// Mitsubishi GX Works2 project: 축   PLC: Q02/Q02H

PROGRAM MAIN
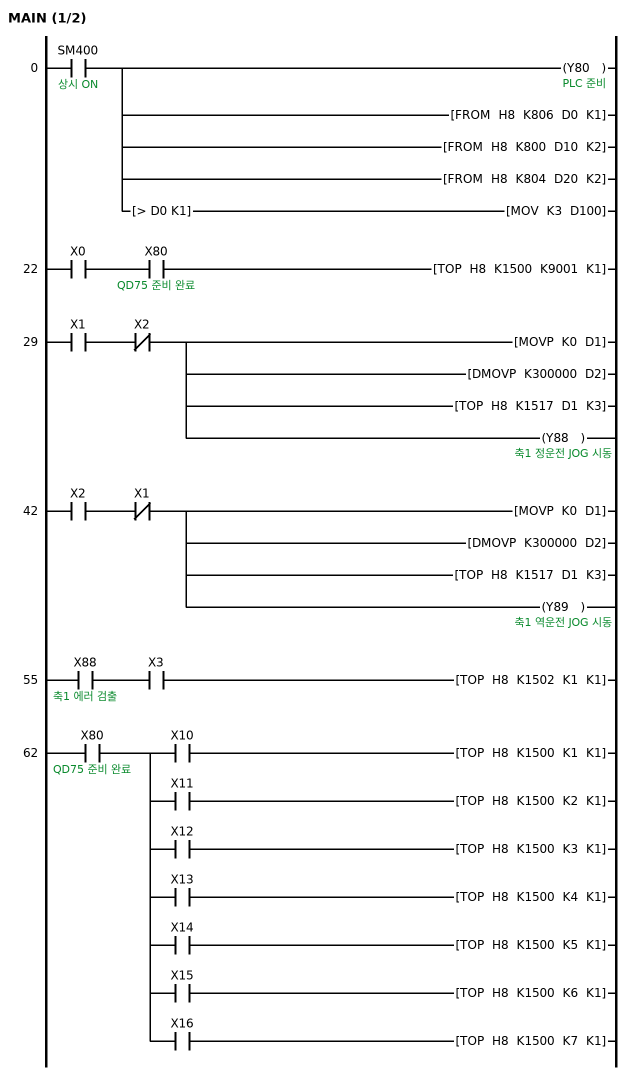
0     LD      SM400  ; 상시 ON
      OUT     Y80  ; PLC 준비
      FROM    H8 K806 D0 K1
      FROM    H8 K800 D10 K2
      FROM    H8 K804 D20 K2
      AND>    D0 K1
      MOV     K3 D100
22    LD      X0
      AND     X80  ; QD75 준비 완료
      TOP     H8 K1500 K9001 K1
29    LD      X1
      ANI     X2
      MOVP    K0 D1
      DMOVP   K300000 D2
      TOP     H8 K1517 D1 K3
      OUT     Y88  ; 축1 정운전 JOG 시동
42    LD      X2
      ANI     X1
      MOVP    K0 D1
      DMOVP   K300000 D2
      TOP     H8 K1517 D1 K3
      OUT     Y89  ; 축1 역운전 JOG 시동
55    LD      X88  ; 축1 에러 검출
      AND     X3
      TOP     H8 K1502 K1 K1
62    LD      X80  ; QD75 준비 완료
      MPS
      AND     X10
      TOP     H8 K1500 K1 K1
      MRD
      AND     X11
      TOP     H8 K1500 K2 K1
      MRD
      AND     X12
      TOP     H8 K1500 K3 K1
      MRD
      AND     X13
      TOP     H8 K1500 K4 K1
      MRD
      AND     X14
      TOP     H8 K1500 K5 K1
      MRD
      AND     X15
      TOP     H8 K1500 K6 K1
      MPP
      AND     X16
      TOP     H8 K1500 K7 K1
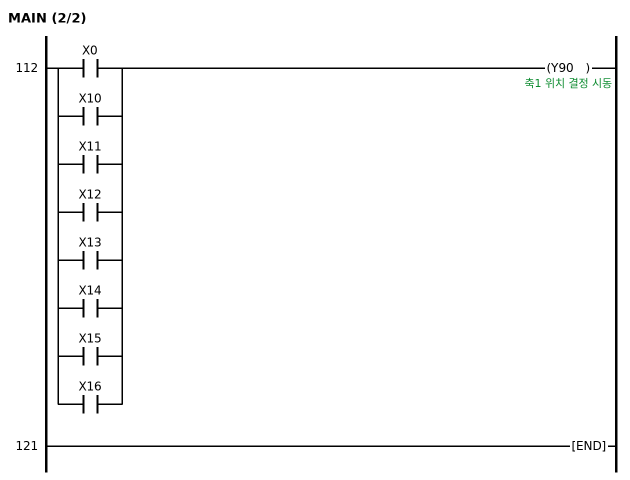
112   LD      X0
      OR      X10
      OR      X11
      OR      X12
      OR      X13
      OR      X14
      OR      X15
      OR      X16
      OUT     Y90  ; 축1 위치 결정 시동
121   END
END_PROGRAM

// device comments not shown above
X81  ; 동기용 플래그
X84  ; 축1 M 코드 ON
X8C  ; 축1 BUSY
X90  ; 축1 시동 완료
X94  ; 축1 위치 결정 완료
Y84  ; 축1 축 정지
Y94  ; 축1 실행 금지 플래그
